TYPE MastLightReq :
STRUCT

RedReq: BOOL;
RedFlashReq: BOOL;
YelReq: BOOL;
YelFlashReq: BOOL;
GrnReq: BOOL;
GrnFlashReq: BOOL;
HornReq: BOOL;	

END_STRUCT
END_TYPE

(* stored: Version 1.1.0.1, ProductVersion 3.1.4024.6
   DUT MastLightReq: Id {17d82285-81cd-4d84-827f-4082bd1af381} *)
